TYPE ST_ValveDeadBand :
STRUCT
	fPosMax : LREAL;
	fPosMin : LREAL;
	fNegMin : LREAL;
	fNegMax : LREAL;
END_STRUCT
END_TYPE

(* stored: Version 1.1.0.1, ProductVersion 3.1.4024.12
   DUT ST_ValveDeadBand: Id {c026af9b-1242-4e36-ac00-a87878b25a19} *)
